Fanuc TP program (LS listing): ALARM_RBT.LS

/PROG  ALARM_RBT
/ATTR
OWNER		= MNEDITOR;
COMMENT		= "";
PROG_SIZE	= 201;
CREATE		= DATE 18-03-06  TIME 14:53:26;
MODIFIED	= DATE 18-03-06  TIME 15:00:30;
FILE_NAME	= ;
VERSION		= 0;
LINE_COUNT	= 1;
MEMORY_SIZE	= 569;
PROTECT		= READ_WRITE;
TCD:  STACK_SIZE	= 0,
      TASK_PRIORITY	= 50,
      TIME_SLICE	= 0,
      BUSY_LAMP_OFF	= 0,
      ABORT_REQUEST	= 0,
      PAUSE_REQUEST	= 0;
DEFAULT_GROUP	= *,*,*,*,*;
CONTROL_CODE	= 00000000 00000000;
/APPL

AUTO_SINGULARITY_HEADER;
  ENABLE_SINGULARITY_AVOIDANCE   : TRUE;

  AUTOZONE_INTERFERENCE_AVOID;
    AUTOZONE_ENABLED         : FALSE;
    AUTOZONE_SCHEDULE_NUMBER : 1;
/MN
   1:  UALM[5] ;
/POS
/END
